FUNCTION_BLOCK FB_LamparaTemporizada_SFC
// La lampara se enciende al accionar el pulsador
// La lampara se apaga transcurrido un tiempo encendida
VAR_INPUT
    TiempoEncendido   : TIME := T#2S;
    IncrementoTiempo  : TIME := T#1S;
END_VAR
VAR_OUTPUT
    TiempoPendiente   : TIME;
END_VAR
VAR
    Lampara   AT %Q*  : BOOL;
    Pulsador  AT %I*  : BOOL;
END_VAR

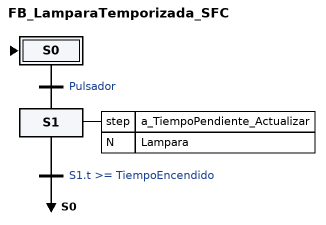
INITIAL_STEP S0:
END_STEP
TRANSITION FROM S0 TO S1
    := Pulsador;
END_TRANSITION
STEP S1:
    a_TiempoPendiente_Actualizar(N);  // step action
    Lampara(N);
END_STEP
TRANSITION FROM S1 TO S0
    := S1.t >= TiempoEncendido;
END_TRANSITION

ACTION a_TiempoPendiente_Actualizar:
TiempoPendiente := TiempoEncendido - S1.t;
END_ACTION

END_FUNCTION_BLOCK

(* stored: Version 1.1.0.1, ProductVersion 3.1.4024.15
   POU FB_LamparaTemporizada_SFC: Id {9fc26670-06c3-48c6-bf53-687a17a3ed03}, SpecialFunc None
   Action a_TiempoPendiente_Actualizar: Id {6203564d-ab62-43c5-974f-a3b810bc5fc3} *)
